(* CODESYS project SFC_TEST.xml

Project tree, tasks and I/O mapping:
  program SFC_TEST [SFC]
*)

// SFC_TEST
PROGRAM SFC_TEST
VAR
	SensorA: BOOL;
	SensorB: BOOL;
END_VAR

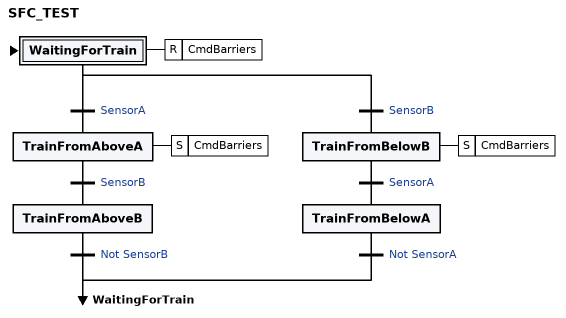
INITIAL_STEP WaitingForTrain:
    CmdBarriers(R);
END_STEP
TRANSITION FROM WaitingForTrain TO TrainFromAboveA
    := SensorA;
END_TRANSITION
STEP TrainFromAboveA:
    CmdBarriers(S);
END_STEP
TRANSITION FROM TrainFromAboveA TO TrainFromAboveB
    := SensorB;
END_TRANSITION
STEP TrainFromAboveB:
END_STEP
TRANSITION FROM TrainFromAboveB TO WaitingForTrain
    := Not SensorB;
END_TRANSITION
TRANSITION FROM WaitingForTrain TO TrainFromBelowB
    := SensorB;
END_TRANSITION
STEP TrainFromBelowB:
    CmdBarriers(S);
END_STEP
TRANSITION FROM TrainFromBelowB TO TrainFromBelowA
    := SensorA;
END_TRANSITION
STEP TrainFromBelowA:
END_STEP
TRANSITION FROM TrainFromBelowA TO WaitingForTrain
    := Not SensorA;
END_TRANSITION

END_PROGRAM
